Universal Robots URScript: custom_0.script

def custom_0():
  global _hidden_verificationVariable=0
  set_tcp(p[0.0,0.0,0.0,0.0,0.0,0.0])
  set_safety_mode_transition_hardness(1)
  motion_version_set(2)
  set_tool_communication(False, 115200, 0, 1, 1.5, 3.5)
  set_tool_output_mode(0)
  set_tool_digital_output_mode(0, 1)
  set_tool_digital_output_mode(1, 1)
  set_tool_voltage(0)
  set_target_payload(1.000000, [0.000000, 0.000000, 0.000000], [0.001539, 0.001539, 0.001539, 0.000000, 0.000000, 0.000000])
  set_gravity([0.0, 0.0, 9.82])
  tool_wrench_limit_disable()
  set_standard_analog_input_domain(0, 1)
  set_standard_analog_input_domain(1, 1)
  set_tool_analog_input_domain(0, 1)
  set_tool_analog_input_domain(1, 1)
  set_analog_outputdomain(0, 0)
  set_analog_outputdomain(1, 0)
  set_input_actions_to_default()
  # begin: URCap Installation Node
  #   Source: External Control, 1.0.5, FZI Research Center for Information Technology
  #   Type: External Control
  # end: URCap Installation Node
  step_count_48f3a27a_0591_49ec_9331_16fca5ce952d = 0.0
  thread Step_Counter_Thread_858ea968_a453_460b_a1ce_90903ced4cf1():
    while (True):
      step_count_48f3a27a_0591_49ec_9331_16fca5ce952d = step_count_48f3a27a_0591_49ec_9331_16fca5ce952d + 1.0
      sync()
    end
  end
  run Step_Counter_Thread_858ea968_a453_460b_a1ce_90903ced4cf1()
  while (True):
    $ 2 "Robot Program"
    # begin: URCap Program Node
    #   Source: External Control, 1.0.5, FZI Research Center for Information Technology
    #   Type: External Control
    $ 3 "Control by 192.168.56.1"
popup("The connection to the remote PC at 192.168.56.1:50002 could not be established. Reason: connect timed out","Receive program failed", False, True, blocking=True)
sync()    # end: URCap Program Node
  end
end
